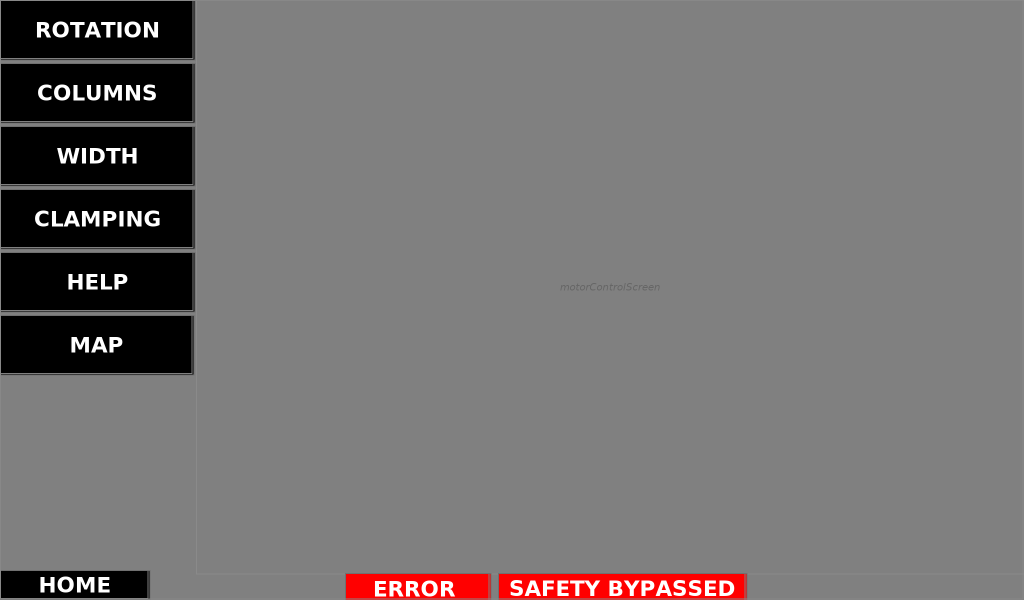
VISUALIZATION multiControlScreen  // 1024x600
    Button (0,570 150x30), "HOME"
        OnMouseDown: change screen: mainScreen
        OnMouseDown: execute { GVL_machine.nPageIndex := 0; GVL_machine.bMotorsInitialized := FALSE; }
    Frame (196,0 829x574), frame switch variable: multiControl.multiCtrlFrameIndex
        shows motorControlScreen()
        shows machineMapScreen()
        shows multiControlHelp()
        shows safetyResetScreen()
        shows tempEflexScreen()
        shows continueAutoScreen()
        shows multiControlHelp()
        shows rotationControl()
        shows widthControl()
    Button (0,0 195x60), "ROTATION", colour toggle: multiControl.nMotorControlIndex = 0
        toggle auto.bResetBtn
        OnMouseDown: execute { multiControl.multiCtrlFrameIndex :=0; multiControl.nMotorControlIndex := 0; }
    Button (498,573 249x31), "SAFETY BYPASSED", invisible if: NOT GVL_machine.bSafetyBypass
        OnMouseDown: change screen: safetyDisableWarning
    Button (345,573 146x32), "ERROR", invisible if: NOT GVL_machine.bDispErrorIcon
        OnMouseDown: change screen: errorScreen
    Button (0,63 195x60), "COLUMNS", colour toggle: multiControl.nMotorControlIndex = 2
        toggle auto.bResetBtn
        OnMouseDown: execute { multiControl.multiCtrlFrameIndex :=0; multiControl.nMotorControlIndex := 2; }
    Button (0,126 195x60), "WIDTH", colour toggle: multiControl.nMotorControlIndex = 3
        toggle auto.bResetBtn
        OnMouseDown: execute { multiControl.multiCtrlFrameIndex :=0; multiControl.nMotorControlIndex := 3; }
    Button (0,189 195x60), "CLAMPING", colour toggle: multiControl.nMotorControlIndex = 1
        toggle auto.bResetBtn
        OnMouseDown: execute { multiControl.multiCtrlFrameIndex :=0; multiControl.nMotorControlIndex := 1; }
    Button (0,252 195x60), "HELP", colour toggle: multiControl.multiCtrlFrameIndex = 2
        toggle auto.bResetBtn
        OnMouseDown: execute { multiControl.multiCtrlFrameIndex := 2; multiControl.nMotorControlIndex := 10; }
    Button (-1,315 195x60), "MAP", colour toggle: multiControl.multiCtrlFrameIndex = 1
        toggle auto.bResetBtn
        OnMouseDown: execute { multiControl.multiCtrlFrameIndex := 1; multiControl.nMotorControlIndex := 10; }
END_VISUALIZATION

(* stored: Version 1.1.0.1, ProductVersion 3.1.4024.13
   Visu multiControlScreen: Id {5a80ee74-77aa-42b2-aa02-3bc33f65ce1d} *)
